FUNCTION_BLOCK WaterSensor
  (* Standard: 61499-2 *)
  (* Version 0.2, 2003-12-04, JHC, Rockwell Automation, Renamed for better indexing. *)
  (* Version 0.1, 2002-11-05, JHC, Rockwell Automation, Corrected missing ST element in Algorithm REQ. *)
  (* Version 0.0, 2000-05-30, JHC, Rockwell Automation *)
  (* Compiler header: package fb.rt.benchmarks.watermonitor; *)
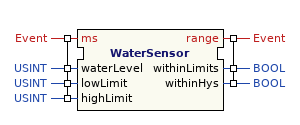
  EVENT_INPUT
    ms WITH waterLevel, lowLimit, highLimit; (* millisecond *)
  END_EVENT
  EVENT_OUTPUT
    range WITH withinLimits, withinHys;
  END_EVENT
  VAR_INPUT
    waterLevel : USINT := 150;
    lowLimit : USINT := 100;
    highLimit : USINT := 200;
  END_VAR
  VAR_OUTPUT
    withinLimits : BOOL := true;
    withinHys : BOOL := true;
  END_VAR
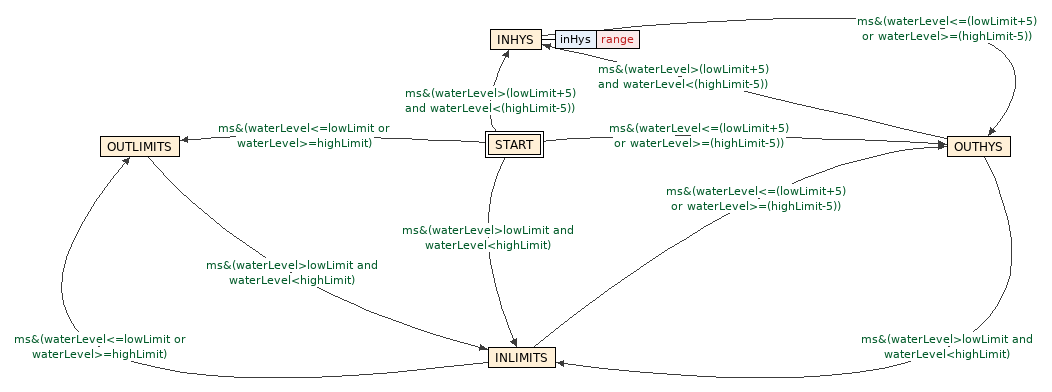
  EC_STATES
    START; (* Initial State *)
    INHYS : inHys -> range; (* in hysterisis *)
    INLIMITS; (* within limts *)
    OUTLIMITS; (* outside limits *)
    OUTHYS; (* outside hysterisis *)
  END_STATES
  EC_TRANSITIONS
    START TO INHYS := ms&(waterLevel>(lowLimit+5) and waterLevel<(highLimit-5));
    START TO OUTHYS := ms&(waterLevel<=(lowLimit+5) or waterLevel>=(highLimit-5));
    START TO INLIMITS := ms&(waterLevel>lowLimit and waterLevel<highLimit);
    START TO OUTLIMITS := ms&(waterLevel<=lowLimit or waterLevel>=highLimit);
    INHYS TO OUTHYS := ms&(waterLevel<=(lowLimit+5) or waterLevel>=(highLimit-5));
    OUTHYS TO INHYS := ms&(waterLevel>(lowLimit+5) and waterLevel<(highLimit-5));
    OUTHYS TO INLIMITS := ms&(waterLevel>lowLimit and waterLevel<highLimit);
    INLIMITS TO OUTHYS := ms&(waterLevel<=(lowLimit+5) or waterLevel>=(highLimit-5));
    INLIMITS TO OUTLIMITS := ms&(waterLevel<=lowLimit or waterLevel>=highLimit);
    OUTLIMITS TO INLIMITS := ms&(waterLevel>lowLimit and waterLevel<highLimit);
  END_TRANSITIONS
  ALGORITHM inHys IN ST: (* Normally executed algorithm *)
withinHys := TRUE;
withinLimits := TRUE;
  END_ALGORITHM
  ALGORITHM outHys IN ST:
withinHys := FALSE;
  END_ALGORITHM
  ALGORITHM inLimits IN ST: (* Initialization algorithm *)
withinLimits := TRUE;
  END_ALGORITHM
  ALGORITHM outLimits IN ST:
withinLimits := FALSE;
withinHys := FALSE;
  END_ALGORITHM
END_FUNCTION_BLOCK
